PROGRAM trigTesting
VAR
END_VAR

END_PROGRAM

(* stored: Version 1.1.0.1, ProductVersion 3.1.4024.11
   POU trigTesting: Id {29ebff99-8be7-45d6-9419-bdb8c4d4b454}, SpecialFunc None *)
